// TwinCAT 3 PLC project PLC1
// ProgramVersion: 3.1.4023.0
// libraries:
//   Tc2_Standard, * (Beckhoff Automation GmbH)
//   Tc2_System, * (Beckhoff Automation GmbH)
//   Tc3_Module, * (Beckhoff Automation GmbH)
// project tree:
//   ControlBox/ FB_ControlBox.TcPOU, G_ControlBox.TcGVL, G_Sim.TcGVL (not stored), E_Status.TcDUT (not stored), FB_Real_Controller.TcPOU, FB_Virtual_Controller.TcPOU, G_IO_Parameters.TcGVL (not stored), G_Virtual_Input.TcGVL, E_Control_Mode.TcDUT (not stored), I_ControlBox.TcIO, ST_Control_Box.TcDUT (not stored)
//   / GlobalTextList.TcGTLO, PlcTask.TcTTO, Visualization Manager.TcVMO (not stored)
//   Programs/ MAIN.TcPOU (not stored), P_ControlBox.TcPOU
//   HMI/ Visualization.TcVIS
// real-time tasks:
//   TASK PlcTask: cycle T#10ms, priority 20, ADS port 350

CONFIGURATION PLC1
    RESOURCE PLC ON TwinCAT3
        TASK PlcTask(INTERVAL := T#10ms, PRIORITY := 20);
        PROGRAM MAIN WITH PlcTask : MAIN;
    END_RESOURCE
END_CONFIGURATION

// ---- ControlBox/G_ControlBox.TcGVL
{attribute 'qualified_only'}
VAR_GLOBAL
	eMode : E_Control_Mode := E_Control_Mode.OFF;
END_VAR

// ---- ControlBox/G_Virtual_Input.TcGVL
{attribute 'qualified_only'}
VAR_GLOBAL
bStart : BOOL := FALSE; // Start button input
bStop : BOOL := FALSE; // Stop button input

bAuto : BOOL := FALSE; // Auto control mode input
bManual : BOOL := FALSE; // Manual control mode input
bOff : BOOL := FALSE; // Off mode

bStopping : BOOL := FALSE;

bJoyActive : BOOL; // Activate the joystick boolean (Top switch)
bJoyNotActive: BOOL; // Inverse logic of JoyActive
fJoyX : REAL := G_IO_Parameters.fMaxInputValue/2 + G_IO_Parameters.fMinInputValue/2; // Variable for storing the joy value in x direction (Cylinder)
fJoyY : REAL := G_IO_Parameters.fMaxInputValue/2 + G_IO_Parameters.fMinInputValue/2; // Variable for storing the joy value in y direction (Winch)
END_VAR

// ---- ControlBox/I_ControlBox.TcIO
INTERFACE I_ControlBox

METHOD Joy_Normalized : REAL
VAR_INPUT
	JoyX_raw : LREAL;
	JoyY_raw : LREAL;
END_VAR
VAR_OUTPUT
	JoyX_normalized : LREAL;
	JoyY_normalized : LREAL;
END_VAR
END_METHOD

METHOD Mode
VAR_OUTPUT
	eMode : E_Control_Mode;
END_VAR
END_METHOD

METHOD Status : E_Status
VAR_OUTPUT
	eStatus : E_Status;
END_VAR
END_METHOD

END_INTERFACE

// ---- ControlBox/FB_ControlBox.TcPOU
FUNCTION_BLOCK FB_ControlBox
VAR_INPUT
	bRealControlBox : BOOL;
END_VAR
VAR_OUTPUT
	eMode : E_Control_Mode;
	eStatus : E_Status;
END_VAR
VAR
	fbVirtualControlBox : FB_Virtual_Controller;
	fbRealControlBox : FB_Real_Controller;
	fbSelectedControlBox : I_ControlBox := fbVirtualControlBox;
END_VAR

IF bRealControlBox THEN
	fbSelectedControlBox := fbRealControlBox;
ELSE
	fbVirtualControlBox.Lamps();
END_IF

fbSelectedControlBox.Mode(eMode => eMode);
fbSelectedControlBox.Status(eStatus => eStatus);
fbSelectedControlBox.Joy_Normalized(fJoyX_raw := G_Virtual_Input.fJoyX, fJoyY_raw := G_Virtual_Input.fJoyY,
									fMin_in := G_IO_Parameters.fMinInputValue, fMax_in := G_IO_Parameters.fMaxInputValue,
									fMin_out := G_IO_Parameters.fMinOutputValue, fMax_out := G_IO_Parameters.fMaxOutputValue,
									fJoyX_normalized => G_Virtual_Input.fJoyX_Normalized, fJoyY_normalized => G_Virtual_Input.fJoyY_Normalized);

END_FUNCTION_BLOCK

// ---- ControlBox/FB_Virtual_Controller.TcPOU
FUNCTION_BLOCK FB_Virtual_Controller IMPLEMENTS I_ControlBox
VAR_INPUT
END_VAR
VAR_OUTPUT
END_VAR
VAR
END_VAR

{warning 'add method implementation '}
METHOD Joy_Normalized : REAL
VAR_INPUT
	// Joy X
	fJoyX_raw : LREAL;
	// Joy Y
	fJoyY_raw : LREAL;
	
	// Min/max in/out parameters
	fMin_in : LREAL;
	fMax_in : LREAL;
	fMin_out : REAL;
	fMax_out : LREAL;
END_VAR
VAR_OUTPUT
	fJoyX_normalized : LREAL;
	fJoyY_normalized : LREAL;
END_VAR

fJoyX_normalized := (fJoyX_raw - fMin_in) * (fMax_out - fMin_out) / (fMax_in - fMin_in) + fMin_out;
fJoyY_normalized := (fJoyY_raw - fMin_in) * (fMax_out - fMin_out) / (fMax_in - fMin_in) + fMin_out;
END_METHOD

METHOD Lamps : REAL
IF G_Virtual_Input.bAuto AND NOT G_Virtual_Input.bManual THEN
	G_Virtual_Input.bAuto := TRUE;
	G_Virtual_Input.bManual := FALSE;
	G_Virtual_Input.bOff := FALSE;
ELSIF G_Virtual_Input.bManual AND NOT G_Virtual_Input.bAuto THEN
	G_Virtual_Input.bAuto := FALSE;
	G_Virtual_Input.bManual := TRUE;
	G_Virtual_Input.bOff := FALSE;
ELSE
	G_Virtual_Input.bAuto := FALSE;
	G_Virtual_Input.bManual := FALSE;
	G_Virtual_Input.bOff := TRUE;
END_IF

IF G_ControlBox.eStatus = E_Status.STOPPING THEN
	G_Virtual_Input.bStopping := TRUE;
ELSE
	G_Virtual_Input.bStopping := FALSE;
END_IF
END_METHOD

{warning 'add method implementation '}
METHOD Mode
VAR_OUTPUT
	eMode : E_Control_Mode;
END_VAR
IF NOT G_Virtual_Input.bAuto AND NOT G_Virtual_Input.bManual AND NOT G_Virtual_Input.bStart THEN
	eMode := E_Control_Mode.OFF;
ELSIF G_Virtual_Input.bAuto AND NOT G_Virtual_Input.bManual AND G_Virtual_Input.bStart THEN
	eMode := E_Control_Mode.AUTO;
ELSIF NOT G_Virtual_Input.bAuto AND G_Virtual_Input.bManual AND G_Virtual_Input.bJoyActive THEN
	eMode := E_Control_Mode.MANUAL;
END_IF
END_METHOD

METHOD Sim
VAR_INPUT
END_VAR
IF G_Virtual_Input.fJoyX_Normalized > 0 AND G_Sim.nX < G_Sim.xMax THEN
	G_Sim.nX := G_Sim.nX+1;
ELSIF G_Virtual_Input.fJoyX_Normalized < 0 AND G_Sim.nX > G_Sim.xMin THEN
	G_Sim.nX := G_Sim.nX-1;
ELSIF G_Virtual_Input.fJoyY_Normalized > 0 AND G_Sim.nY < G_Sim.yMax THEN
	G_Sim.nY := G_Sim.nY+1;
ELSIF G_Virtual_Input.fJoyY_Normalized < 0 AND G_Sim.nY > G_Sim.yMin THEN
	G_Sim.nY := G_Sim.nY-1;
END_IF
END_METHOD

{warning 'add method implementation '}
METHOD Status : E_Status
VAR_OUTPUT
	eStatus : E_Status;
END_VAR
IF G_ControlBox.eMode = E_Control_Mode.OFF THEN
	eStatus := E_Status.NOTREADY;
END_IF
IF G_ControlBox.eMode = E_Control_Mode.MANUAL OR G_ControlBox.eMode = E_Control_Mode.AUTO THEN
	eStatus := E_Status.READY;
END_IF
IF G_Virtual_Input.bStart THEN
	eStatus := E_Status.STARTING;
END_IF
IF (G_ControlBox.eMode = E_Control_Mode.MANUAL AND G_Virtual_Input.bStart) OR (G_ControlBox.eMode = E_Control_Mode.AUTO AND G_Virtual_Input.bStart) THEN
	eStatus := E_Status.RUNNING;
END_IF
IF G_Virtual_Input.bStop THEN
	eStatus := E_Status.STOPPING;
END_IF
END_METHOD

END_FUNCTION_BLOCK

// ---- ControlBox/FB_Real_Controller.TcPOU
FUNCTION_BLOCK FB_Real_Controller IMPLEMENTS I_ControlBox
VAR_INPUT
END_VAR
VAR_OUTPUT
END_VAR
VAR
END_VAR

{warning 'add method implementation '}
METHOD Joy_Normalized : REAL
VAR_INPUT
	JoyX_raw	: LREAL;
	JoyY_raw	: LREAL;
END_VAR
VAR_OUTPUT
	JoyX_normalized	: LREAL;
	JoyY_normalized	: LREAL;
END_VAR
END_METHOD

{warning 'add method implementation '}
METHOD Mode
VAR_OUTPUT
	eMode	: E_Control_Mode;
END_VAR
END_METHOD

{warning 'add method implementation '}
METHOD Status : E_Status
VAR_OUTPUT
	eStatus : E_Status;
END_VAR
END_METHOD

END_FUNCTION_BLOCK

// ---- Programs/P_ControlBox.TcPOU
PROGRAM P_ControlBox
VAR
	fbControlBox : FB_ControlBox;
END_VAR

fbControlBox(bRealControlBox := FALSE, eMode => G_ControlBox.eMode); // Run controlbox FB with argument. If bRealControlBox is TRUE, then the FB_RealControlBox will be selected when running the program.

END_PROGRAM

// ---- GlobalTextList.TcGTLO
TEXTLIST GlobalTextList
  344 = '%f'
  126 = '%s'
  129 = '+'
  960 = '-'
  359 = 'Activate joy'
  818 = 'AUTO'
  882 = 'Control'
  803 = 'Control box'
  27 = 'Controller'
  247 = 'Fancy Pancy controller 0.0001'
  914 = 'Joy top switch'
  836 = 'Joy X'
  464 = 'Joy Y'
  849 = 'Label'
  236 = 'MANUAL'
  890 = 'Mode:'
  833 = 'Start'
  776 = 'Status:'
  326 = 'Stop'
  589 = 'X'
  907 = 'X:'
  335 = 'Y:'
END_TEXTLIST

// ---- HMI/Visualization.TcVIS
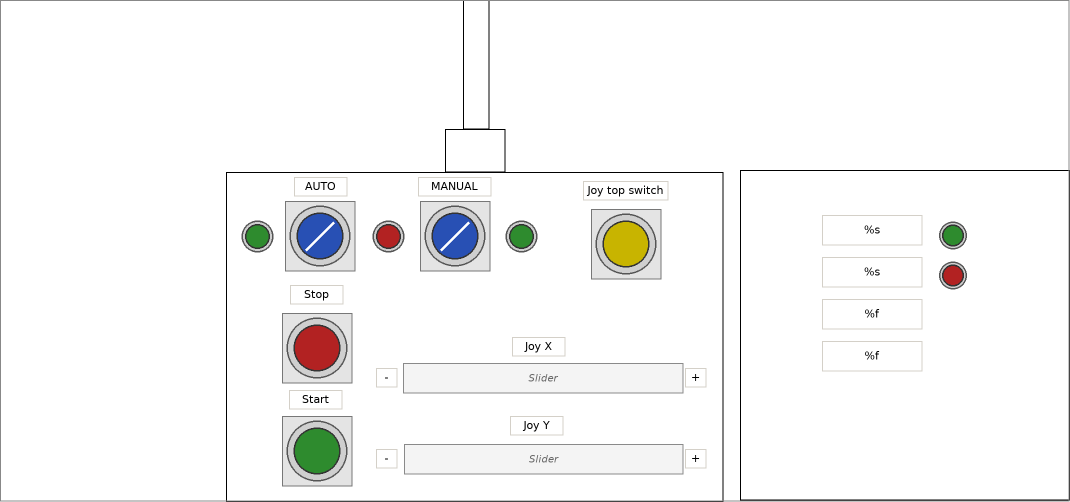
VISUALIZATION Visualization  // 1070x502
    RoundedRectangle (226,172 497x330)
    RotarySwitch (285,201 70x70), variable: G_Virtual_Input.bAuto, behaviour: TOGGLE, style: Switch-RotarySwitch-Blue
    PushSwitch (282,416 70x70), variable: G_Virtual_Input.bStart, behaviour: TOGGLE, style: Switch-PushSwitch-Green
    PushSwitch (282,313 70x70), variable: G_Virtual_Input.bStop, behaviour: TOGGLE, style: Switch-PushSwitch-Red
    RotarySwitch (420,201 70x70), variable: G_Virtual_Input.bManual, behaviour: TOGGLE, style: Switch-RotarySwitch-Blue
    Slider (404,444 279x30), variable: G_Virtual_Input.fJoyY, input disabled if: G_Virtual_Input.bJoyNotActive, scale 0..0
    Slider (403,363 280x30), variable: G_Virtual_Input.fJoyX, input disabled if: G_Virtual_Input.bJoyNotActive, scale 0..0
    Rectangle (445,129 60x43)
    Rectangle (463,0 26x129)
    Textfield (290,285 53x19), "Stop"
    Textfield (289,390 53x19), "Start"
    Textfield (512,337 53x19), "Joy X"
    Textfield (510,416 53x19), "Joy Y"
    PushSwitchLed (591,209 70x70), variable: G_Virtual_Input.bJoyActive, behaviour: TOGGLE, style: Switch-PushSwitchLed-Yellow
    Textfield (583,181 85x19), "Joy top switch"
    Textfield (685,368 21x19), "+"
    Textfield (685,449 21x19), "+"
    Textfield (376,449 21x19), "-"
    Textfield (376,368 21x19), "-"
    Textfield (294,177 53x19), "AUTO"
    Textfield (418,177 73x19), "MANUAL"
    RoundedRectangle (740,170 330x330)
    Label (756,214 63x30), "Mode:"
    Label (738,253 90x38), "Status:"
    Textfield (822,215 100x30), "%s", text variable: G_ControlBox.eMode
    Lamp1 (937,215 32x41), style: Lamp-Lamp1-Green
    Textfield (822,257 100x30), "%s", text variable: G_ControlBox.eStatus
    Lamp1 (937,255 32x41), variable: G_Virtual_Input.bStopping, style: Lamp-Lamp1-Red
    Lamp1 (239,216 37x41), variable: G_Virtual_Input.bAuto, style: Lamp-Lamp1-Green
    Lamp1 (370,216 37x41), variable: G_Virtual_Input.bOff, style: Lamp-Lamp1-Red
    Lamp1 (503,216 37x41), variable: G_Virtual_Input.bManual, style: Lamp-Lamp1-Green
    Textfield (822,299 100x30), "%f", text variable: G_Virtual_Input.fJoyX_Normalized
    Textfield (822,341 100x30), "%f", text variable: G_Virtual_Input.fJoyY_Normalized
    Label (780,298 45x38), "X:"
    Label (780,337 45x38), "Y:"
END_VISUALIZATION
